Fanuc TP program (LS listing): RECSTEPA.LS

/PROG  RECSTEPA
/ATTR
OWNER		= MNEDITOR;
COMMENT		= "RecStepA";
PROG_SIZE	= 0;
CREATE		= DATE 26-01-01  TIME 00:00:00;
MODIFIED	= DATE 26-01-01  TIME 00:00:00;
FILE_NAME	= ;
VERSION		= 0;
LINE_COUNT	= 4;
MEMORY_SIZE	= 0;
PROTECT		= READ_WRITE;
TCD:  STACK_SIZE	= 0,
      TASK_PRIORITY	= 50,
      TIME_SLICE	= 0,
      BUSY_LAMP_OFF	= 0,
      ABORT_REQUEST	= 0,
      PAUSE_REQUEST	= 0;
DEFAULT_GROUP	= 1,*,*,*,*;
CONTROL_CODE	= 00000000 00000000;
/MN
   1:  !RAPID RecordProbe.RecStepA ;
   2:  R[2:recCtrl.state]=1    ;
   3:  R[1:recCtrl.counter]=R[1:recCtrl.counter]+1    ;
   4:  F[1]=(ON) ;
/POS
/END
